{attribute addProperty BoxType "KL6224-0003"}
{attribute addProperty Id "Channel_1Channel_0418AA5000"}
{attribute addProperty CRC "3328131575"}
{attribute addProperty SizeInBites "0"}
{attribute addProperty SizeInBytes "0"}
TYPE KL_C65F41F7 :
STRUCT
	{attribute addProperty Name "Channel_1"}
	Channel_1 : Channel_0418AA50;
END_STRUCT
END_TYPE

(* stored: Version 1.2.0.0, ProductVersion 3.1.4024.9
   DUT KL_C65F41F7: Id {626d0965-cfc4-40da-bd02-2c0a18b30f77} *)
